/// This struct contains variables that
/// * are read from outside (e.g. HMI) to retrieve information about the unit's current state and (temporary) parameters (= `publish`) 
/// * are written from outside (e.g. HMI) to control the unit via ADS (= `subscribe`) 
TYPE ScriblyCom :
STRUCT
  Publish : ScriblyComPublish;
  Subscribe : ScriblyComSubscribe;
END_STRUCT
END_TYPE

(* stored: Version 1.1.0.1
   DUT ScriblyCom: Id {420ddea8-f42e-4032-9829-11ba88780de4} *)
